(* CODESYS project CtaSysBase_1.0.0.0.library
   Description: Basis Library der CTA
   Version: 1.0.0.0
   Title: CtaSysBase
   Author: SIS
   Company: CTA
   Placeholder: CtaSysBase
   DocFormat: reStructuredText
   DefaultNamespace: CtaSysBase
   CompiledLibraryCompatibilityVersion: CODESYS V3.5 SP16 Patch 3
   LanguageModelAttribute: qualified-access-only

Project tree, tasks and I/O mapping:
  libraries: VisuSymbols, 4.5.0.0 (System); CtaVisSymbols, 1.0.0.0 (CTA); CtaVisHelp, 1.0.0.0 (CTA)
  40 Visualizations/
  30 Program Organization Units/
    function block fbBASE [ST]: proGetInstancePath, proSetInstancePath
  00000000-0000-0000-0000-000000000000|D:\CoDeSys\LibrariesV3\trunk\Intern\CAA\CAA Template\3.4.0.0 draft\Placeholder.xml
  00000000-0000-0000-0000-000000000000|D:\CoDeSys\LibrariesV3\trunk\Intern\CAA\CAA Template\3.2.0.3 draft\Prefix.pdf
  00000000-0000-0000-0000-000000000000|D:\CoDeSys\LibrariesV3\trunk\Intern\CAA\CAA Template\3.5.2.0 draft\Placeholder.xml
  20 Structs/
  50 Images/
  10 Documenation/
    global variables VersionHistory
    global variables readMe
  21 Interface/
    interface ITF_BASE: proGetInstancePath, proSetInstancePath
  11 Library Parameter/
  12 Konstanten/
  60 Textlisten/
  13 Globale Variablen/
*)

// 10 Documenation/VersionHistory
(* 

.. image:: ../../Images/CTA_Logo.jpg
   :align: right
   :width: 15% 

**Vorlage**   


============ =========== =========== ============================================
**Date**     **Version** **Author**  **Change**
------------ ----------- ----------- --------------------------------------------
04.03.2021   0.0.0.0     SIS         Vorlage erstellt

============ =========== =========== ============================================


*)
VAR_GLOBAL
    stInfo : STRING:= '0.0.0.0, Vorlage, CTA';
END_VAR

// 10 Documenation/readMe
(*

**ReadMe**
 
|	**Empfehlung**
|
|	Dokumentrieren Sie die Library für eine nachhaltige Entwicklung
|     
| *Beispiel* 
|
| Dies ist die Vorlage Library der CTA. Erstellen Sie ihre Library anhand dieser Vorlage.
*)

VAR_GLOBAL
    xReadMeDone              :   BOOL;
END_VAR

// 21 Interface/ITF_BASE
(*Base Interface single Responsibility Instance Name*)
INTERFACE ITF_BASE EXTENDS __SYSTEM.IQueryInterface

(*Get Instance Name *)
PROPERTY proGetInstancePath : STRING[255]
GET
END_GET
END_PROPERTY

PROPERTY proSetInstancePath : STRING[255]
SET
END_SET
END_PROPERTY

END_INTERFACE

// 30 Program Organization Units/fbBASE
(*Base Functionblock single Responsibility Instance Name*)
{attribute 'reflection'}
{attribute 'enable_dynamic_creation'}
FUNCTION_BLOCK fbBASE IMPLEMENTS ITF_BASE
VAR
	{attribute 'instance-path'}
	{attribute 'noinit'}
	{attribute 'monitoring_encoding' := 'UTF-8'}
	stInstancePath	: STRING[255];
END_VAR

///Get Instance Name 
PROPERTY proGetInstancePath : STRING[255]
GET
proGetInstancePath := stInstancePath;
END_GET
END_PROPERTY

PROPERTY proSetInstancePath : STRING[255]
SET
stInstancePath := proSetInstancePath;
END_SET
END_PROPERTY

END_FUNCTION_BLOCK
